FUNCTION_BLOCK FB_Light
VAR_INPUT
END_VAR
VAR_OUTPUT
END_VAR
VAR
	bIsOn	:BOOL;
END_VAR

METHOD turnLightOff : BOOL
VAR_INPUT
END_VAR
ADSLOGSTR(msgCtrlMask:= ADSLOG_MSGTYPE_ERROR, msgFmtStr:= 'Light is off', strArg:= '');
bIsOn := FALSE;
END_METHOD

METHOD turnLightOn : BOOL
VAR_INPUT
END_VAR
ADSLOGSTR(msgCtrlMask:= ADSLOG_MSGTYPE_ERROR, msgFmtStr:= 'Light is on', strArg:= '');
bIsOn := TRUE;
END_METHOD

END_FUNCTION_BLOCK

(* stored: Version 1.1.0.1
   POU FB_Light: Id {84668e9a-79dd-49d1-a8d0-e22b0ab3419f}, SpecialFunc None
   Method turnLightOff: Id {cdc6f5ba-67c7-4fc7-9b0e-91eca7d205fa}
   Method turnLightOn: Id {1de21c0e-d2c3-4af7-ace3-0be53d378cc1} *)
